PROGRAM PRG_TEST
VAR
END_VAR

END_PROGRAM

(* stored: Version 1.1.0.1, ProductVersion 3.1.4024.11
   POU PRG_TEST: Id {b0b9f2e5-28eb-44e0-8846-21a78d2e9989}, SpecialFunc None *)
